{attribute addProperty BoxType "EK1100-0000-0018"}
{attribute addProperty Id "Beckhoff_AX88xxEK1122Beckhoff_AX88xxEK1122_27E1F918162A_0001_AX8810_0000_0017AX8810_B7ACDB9016220.25A_0002_AX8810_0000_0024AX8810_4A92314216220.25A_0003_AX8810_0000_0100AX8810_4A92314216220.25"}
{attribute addProperty CRC "1468131005"}
{attribute addProperty SizeInBites "502"}
{attribute addProperty SizeInBytes "62.75"}
TYPE Beckhoff_AX88xx_5781E6BD EXTENDS EK1100_179A0949 :
STRUCT
	{attribute addProperty Name "Beckhoff_AX88xxEK1122"}
	Beckhoff_AX88xxEK1122 : Beckhoff_AX88xxEK1122_27E1F918;
	{attribute addProperty Name "A_0001_AX8810_0000_0017"}
	A_0001_AX8810_0000_0017 : AX8810_B7ACDB90;
	{attribute addProperty Name "A_0002_AX8810_0000_0024"}
	A_0002_AX8810_0000_0024 : AX8810_4A923142;
	{attribute addProperty Name "A_0003_AX8810_0000_0100"}
	A_0003_AX8810_0000_0100 : AX8810_4A923142;
END_STRUCT
END_TYPE

(* stored: Version 1.2.0.0, ProductVersion 3.1.4024.9
   DUT Beckhoff_AX88xx_5781E6BD: Id {513d0d75-65fd-4186-89ad-65763656a4ed} *)
